// TIA Portal V19 export
TYPE "UDT_STATUS_SIM"
   STRUCT
      out : Bool;
      actual : Bool;
      simulated : Bool;
      simValue : Bool;
   END_STRUCT;
END_TYPE
